// TIA Portal V21 export
FUNCTION "Main consensi" : Void   // FC70, LAD
{ S7_Optimized_Access := 'TRUE' }
// stored: SetENOAutomatically false
   VAR_TEMP
      TotalizzatoreOltreMetà : Bool;
      OutSegnale : Bool;
      SegnaleDaInviare : Bool;
   END_VAR
BEGIN
END_FUNCTION
